# EPICS autosave request: iocBoot/iocSoftGlueZynq/SGMenu.req
file configMenu.req P=$(P),CONFIG=$(CONFIG)
file softGlue_settings.req  P=$(P),H=$(H)
